(* IEC 61131-3 sources: RL_MAR/experiments/comparison/autoplc/results/deepseek-ai-DeepSeek-V3.2_20260508_111905/med_25, 1 file *)

(* ---- med_25_1.st ---- *)
FUNCTION_BLOCK WastewaterControl
VAR_INPUT
    InFlow : REAL;
    OutFlow : REAL;
    pH : REAL;
    TankLvl : REAL;
END_VAR

VAR_OUTPUT
    Pump1 : BOOL;
    Pump2 : BOOL;
    Valve1 : BOOL;
    Valve2 : BOOL;
END_VAR

VAR
    LowInFlow : REAL := 100.0;
    HighOutFlow : REAL := 90.0;
    DesiredPH : REAL := 7.0;
    HighTankLvl : REAL := 80.0;
END_VAR

// Main control logic
// Evaluate Pump1 condition
IF InFlow < LowInFlow THEN
    Pump1 := TRUE;
ELSE
    Pump1 := FALSE;
END_IF;

// Evaluate Pump2 condition
IF OutFlow > HighOutFlow THEN
    Pump2 := TRUE;
ELSE
    Pump2 := FALSE;
END_IF;

// Evaluate Valve1 condition
IF pH < DesiredPH THEN
    Valve1 := TRUE;
ELSE
    Valve1 := FALSE;
END_IF;

// Evaluate Valve2 condition
IF TankLvl > HighTankLvl THEN
    Valve2 := TRUE;
ELSE
    Valve2 := FALSE;
END_IF;

END_FUNCTION_BLOCK
